// TIA Portal project "RollerConveyorSimulatorUc" (V17)
// Vorlageprojekt für das Buch mit Zielsystem S7-1200

(* hardware
DEVICE "S7-1200-Station_1"  S7-1200 Station
   slot 0: "Baugruppenträger_0"  Rack  V1.0
   slot 1: "PLC_1"  CPU 1211C DC/DC/DC  6ES7 211-1AE40-0XB0  V4.1
*)

// ===== PLC "PLC_1"  CPU 1211C DC/DC/DC =====

VAR_GLOBAL   // PLC tag table "Standard-Variablentabelle"
   "Tag_1" AT %A0.0 : Bool;
   "Tag_2" AT %E0.0 : Bool;
   "Tag_3" AT %E0.1 : Bool;
   "ACİL STOP" AT %I15.0 : Bool;
   "Tag_5" AT %M0.2 : Bool;
   "3.NOLU KONVEYOR" AT %Q12.2 : Bool;
   "START" AT %I15.1 : Bool;
   "2.NOLU KONVEYOR" AT %Q12.1 : Bool;
   "Tag_6" AT %M0.1 : Bool;
   "Tag_4" AT %M10.0 : Bool;
   "Tag_7" AT %M0.0 : Bool;
   "1.NOLU KONVEYOR" AT %Q12.0 : Bool;
   "STOP" AT %I15.2 : Bool;
END_VAR

// folder: System blocks/Program resources

DATA_BLOCK "IEC_Timer_0_DB"   // DB1
{ S7_Optimized_Access := 'TRUE' }
AUTHOR : Simatic
FAMILY : IEC
NAME : IEC_TMR
VERSION : 1.0
// stored: InstanceOfName IEC_TIMER
"IEC_TIMER"
BEGIN
END_DATA_BLOCK

DATA_BLOCK "IEC_Timer_0_DB_1"   // DB2
{ S7_Optimized_Access := 'TRUE' }
AUTHOR : Simatic
FAMILY : IEC
NAME : IEC_TMR
VERSION : 1.0
// stored: InstanceOfName IEC_TIMER
"IEC_TIMER"
BEGIN
END_DATA_BLOCK

DATA_BLOCK "IEC_Timer_0_DB_2"   // DB3
{ S7_Optimized_Access := 'TRUE' }
AUTHOR : Simatic
FAMILY : IEC
NAME : IEC_TMR
VERSION : 1.0
// stored: InstanceOfName IEC_TIMER
"IEC_TIMER"
BEGIN
END_DATA_BLOCK

DATA_BLOCK "IEC_Timer_0_DB_3"   // DB4
{ S7_Optimized_Access := 'TRUE' }
AUTHOR : Simatic
FAMILY : IEC
NAME : IEC_TMR
VERSION : 1.0
// stored: InstanceOfName IEC_TIMER
"IEC_TIMER"
BEGIN
END_DATA_BLOCK

// folder: (top level)

FUNCTION "MHJ-PLC-Lab-Function-S71200" : Void   // FC9000, SCL
{ S7_Optimized_Access := 'TRUE' }
VERSION : 0.1
   VAR_TEMP
      rdTimeReturn : Int;
      outputTime : DTL;
      SyncVal : Byte;
      forVal : Int;
      forVal_2 : Int;
      Value : Byte;
   END_VAR
   VAR CONSTANT
      CompVal : Byte := 16#34;
      Value_01 : Byte := 16#11;
      Value_01_DW : DWord := 16#A165_D992;
      Value_02_DW : DWord := 16#58BE_4401;
   END_VAR
BEGIN

   #Value:=PEEK(area := 16#82,
        dbNumber := 0,
        byteOffset := 511);
   #Value := #Value + 1;

   POKE(area := 16#82,
        dbNumber := 0,
        byteOffset := 511,
        value := #Value);

   POKE(area:=16#81,
        dbNumber:=0,
        byteOffset:=1016,
        value:=#Value_01_DW);
   POKE(area := 16#81,
        dbNumber := 0,
        byteOffset := 1020,
        value := #Value_02_DW);

   POKE(area := 16#81,
        dbNumber := 0,
        byteOffset := 511,
        value := B#16#00);

   FOR #forVal := 0 TO 120 DO
       FOR #forVal_2:=0 TO 10 DO
           #rdTimeReturn:=RD_SYS_T(#outputTime);
           #rdTimeReturn := WR_SYS_T(#outputTime);
           #rdTimeReturn := RD_SYS_T(#outputTime);
           #rdTimeReturn := WR_SYS_T(#outputTime);
       END_FOR;
       #SyncVal:= PEEK(area := 16#81,
                      dbNumber := 0,
                      byteOffset := 511);
       IF #SyncVal = #CompVal THEN
          GOTO M_1;
       END_IF;
   END_FOR;
   RETURN;

   M_1:
   POKE(area := 16#81,
        dbNumber := 0,
        byteOffset := 511,
        value := B#16#0);
END_FUNCTION

ORGANIZATION_BLOCK "Main"   // OB1, LAD, ProgramCycle
TITLE = "Main Program Sweep (Cycle)"
{ S7_Optimized_Access := 'TRUE' }
VERSION : 0.1
   VAR_INPUT
      Initial_Call : Bool;   // Initial call of this OB
      Remanence : Bool;   // =True, if remanent data are available
   END_VAR
BEGIN

REGION Network 1: Konnektierungsbaustein für PLC-Lab
   // Im Netzwerk 1 wird der Konnektierungsbaustein für PLC-Lab aufgerufen.
   // Dieser Aufruf darf nicht entfernt werden!
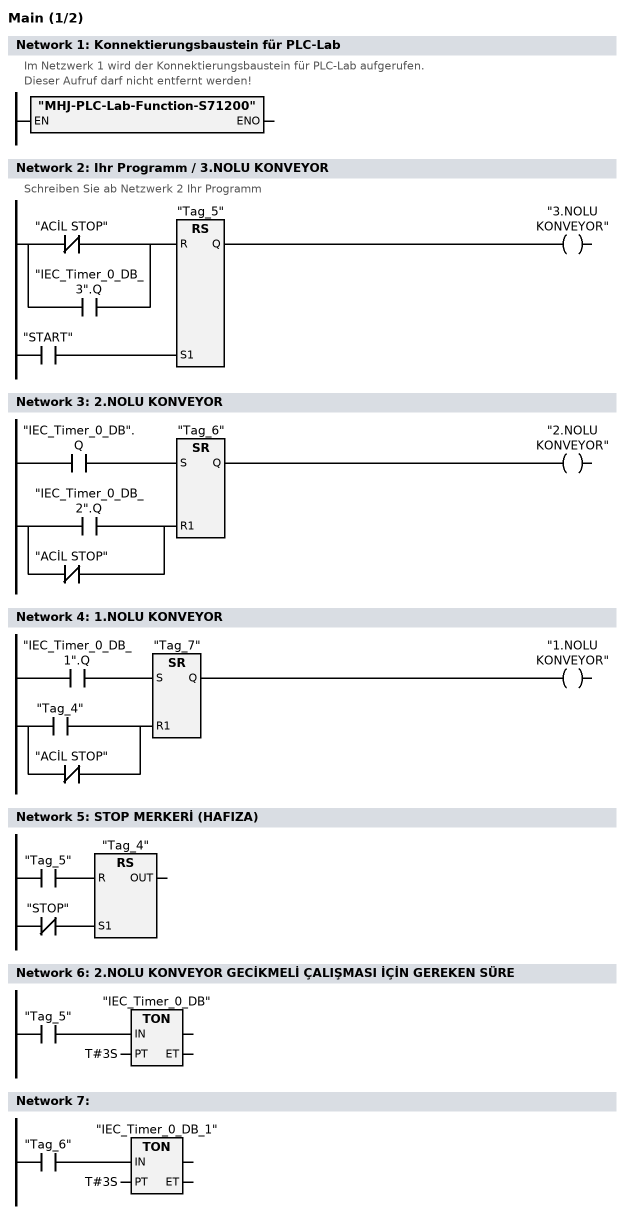
   RUNG wire#powerrail
      "MHJ-PLC-Lab-Function-S71200"()
   END_RUNG
   // the same network as SCL:
   "MHJ-PLC-Lab-Function-S71200"();
END_REGION

REGION Network 2: Ihr Programm / 3.NOLU KONVEYOR
   // Schreiben Sie ab Netzwerk 2 Ihr Programm
   RUNG wire#powerrail
      I_Contact( "ACİL STOP" )
      wire#w1
      S_RS(operand := "Tag_5", s1 := wire#w2)
      Coil( "3.NOLU KONVEYOR" )
   END_RUNG
   RUNG wire#powerrail
      Contact( "IEC_Timer_0_DB_3".Q )
   END_RUNG wire#w1
   RUNG wire#powerrail
      Contact( "START" )
   END_RUNG wire#w2
   // the same network as SCL:
   IF NOT "ACİL STOP" OR "IEC_Timer_0_DB_3".Q THEN
       "Tag_5" := FALSE;   // RS flip-flop
   END_IF;
   IF "START" THEN "Tag_5" := TRUE; END_IF;
   "3.NOLU KONVEYOR" := "Tag_5";
END_REGION

REGION Network 3: 2.NOLU KONVEYOR
   RUNG wire#powerrail
      Contact( "IEC_Timer_0_DB".Q )
      S_SR(operand := "Tag_6", r1 := wire#w1)
      Coil( "2.NOLU KONVEYOR" )
   END_RUNG
   RUNG wire#powerrail
      Contact( "IEC_Timer_0_DB_2".Q )
   END_RUNG wire#w1
   RUNG wire#powerrail
      I_Contact( "ACİL STOP" )
   END_RUNG wire#w1
   // the same network as SCL:
   IF "IEC_Timer_0_DB".Q THEN
       "Tag_6" := TRUE;   // SR flip-flop
   END_IF;
   IF "IEC_Timer_0_DB_2".Q OR NOT "ACİL STOP" THEN "Tag_6" := FALSE; END_IF;
   "2.NOLU KONVEYOR" := "Tag_6";
END_REGION

REGION Network 4: 1.NOLU KONVEYOR
   RUNG wire#powerrail
      Contact( "IEC_Timer_0_DB_1".Q )
      S_SR(operand := "Tag_7", r1 := wire#w1)
      Coil( "1.NOLU KONVEYOR" )
   END_RUNG
   RUNG wire#powerrail
      Contact( "Tag_4" )
   END_RUNG wire#w1
   RUNG wire#powerrail
      I_Contact( "ACİL STOP" )
   END_RUNG wire#w1
   // the same network as SCL:
   IF "IEC_Timer_0_DB_1".Q THEN
       "Tag_7" := TRUE;   // SR flip-flop
   END_IF;
   IF "Tag_4" OR NOT "ACİL STOP" THEN "Tag_7" := FALSE; END_IF;
   "1.NOLU KONVEYOR" := "Tag_7";
END_REGION

REGION Network 5: STOP MERKERİ (HAFIZA)
   RUNG wire#powerrail
      Contact( "Tag_5" )
      S_RS(operand := "Tag_4", s1 := wire#w1)
   END_RUNG
   RUNG wire#powerrail
      I_Contact( "STOP" )
   END_RUNG wire#w1
   // the same network as SCL:
   IF "Tag_5" THEN
       "Tag_4" := FALSE;   // RS flip-flop
   END_IF;
   IF NOT "STOP" THEN "Tag_4" := TRUE; END_IF;
END_REGION

REGION Network 6: 2.NOLU KONVEYOR GECİKMELİ ÇALIŞMASI İÇİN GEREKEN SÜRE
   "IEC_Timer_0_DB".TON(IN := "Tag_5", PT := T#3S);
END_REGION

REGION Network 7
   "IEC_Timer_0_DB_1".TON(IN := "Tag_6", PT := T#3S);
END_REGION

REGION Network 8
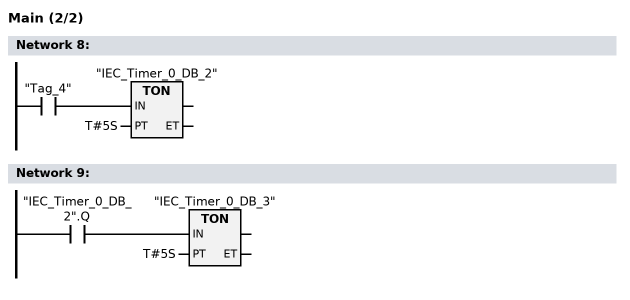
   "IEC_Timer_0_DB_2".TON(IN := "Tag_4", PT := T#5S);
END_REGION

REGION Network 9
   "IEC_Timer_0_DB_3".TON(IN := "IEC_Timer_0_DB_2".Q, PT := T#5S);
END_REGION
END_ORGANIZATION_BLOCK